// TIA Portal V19 export
DATA_BLOCK "JB"   // DB52
// stored: InstanceOfName JB_FB, InstanceOfType FB
"JB_FB"
   // VAR_INPUT
   //    AreaInterface : "AreaInterface";
   //    ZSI : "udt_ZoneSafetyInterface";
   //    DSI : Struct
   //       Torch : "udt_DeviceSafetyInterface";
   //       ClampEntry : "udt_DeviceSafetyInterface";
   //       ClampExit : "udt_DeviceSafetyInterface";
   //       CutHead : "udt_DeviceSafetyInterface";
   //       PinchRoll_Feed : "udt_DeviceSafetyInterface";
   //       PinchRoll_Lift : "udt_DeviceSafetyInterface";
   //    END_STRUCT;
   //    Drive : Struct
   //       Torch : "TAx_DriveInterface";
   //       Picnhroll_Feed : "TAx_DriveInterface";
   //    END_STRUCT;
   //    HWID : Struct
   //       Torch_TEL1 : HW_SUBMODULE;
   //       TorchEnc_IO : HW_SUBMODULE;
   //       Pinchroll_Feed_TEL1 : HW_SUBMODULE;
   //    END_STRUCT;
   //    DataIn : Struct
   //       WeldingCycle_AI_Potentiometer : Int;
   //       WeldingCycle_Pb_Stop : Bool;
   //       WeldingCycle_Pb_Start : Bool;
   //       WeldingCycle_Pb_StartStop : Bool;
   //       Welder_Pb_Man : Bool;
   //       CutHead_PbCycle : Bool;
   //       SAFETY_DeadMan_PB : Bool;
   //       Torch : "Positioning_DOL_Machine_DataIn";
   //       ClampEntry : "ValveMachine_DataIn";
   //       ClampExit : "ValveMachine_DataIn";
   //       CutHead : "ValveMachine_DataIn";
   //       PinchRoll_Feed : "SpeedMachine_DataIn";
   //       PinchRoll_Lift : "ValveMachine_DataIn";
   //    END_STRUCT;
   //    CIn : Struct
   //       Manager : "JB_Manager";
   //       PressureRunning : Bool;
   //    END_STRUCT;
   //    Config : Struct
   //       MeasurePasslineReference : Real;
   //       MaxMaterialWidth : Real;
   //       Torch : "Positioning_DOL_Machine_Config";
   //       ClampEntry : "ValveMachine_Config";
   //       ClampExit : "ValveMachine_Config";
   //       CutHead : "ValveMachine_Config";
   //       Pinchroll_Feed : "SpeedMachine_Config";
   //       Pinchroll_Lift : "ValveMachine_Config";
   //    END_STRUCT;
   // END_VAR
   // VAR_OUTPUT
   //    MachineInterface : "MachineInterface";
   //    DataOut : Struct
   //       LpWeldingCycle_1 : Bool;
   //       LpWeldingCycle_2 : Bool;
   //       WelderON : Bool;
   //       AspiratoreON : Bool;
   //       Torch : "Positioning_DOL_Machine_DataOut";
   //       ClampEntry : "ValveMachine_DataOut";
   //       ClampExit : "ValveMachine_DataOut";
   //       CutHead : "ValveMachine_DataOut";
   //       Pinchroll_Feed : "SpeedMachine_DataOut";
   //       Pinchroll_Lift : "ValveMachine_DataOut";
   //    END_STRUCT;
   //    COut : "JB_Status";
   // END_VAR
   // VAR_IN_OUT
   //    PersistentValues : Struct
   //       Data : Struct
   //          WeldingSetUp : "JB_WeldingSetUp";
   //          ClampEntryClosed : Bool;
   //          ClampExitClosed : Bool;
   //       END_STRUCT;
   //       Torch : Struct
   //          MeasureTorchHolder : LReal;
   //          InhibitWeld_Pos : LReal;
   //          InhibitWeld_Window : LReal;
   //          Parking_Pos : LReal;
   //          WeldingUseLocalData : Bool;
   //          Cycle_HighSpeed : LReal;
   //          Cycle_LowSpeed : LReal;
   //       END_STRUCT;
   //       TorchAx : "Positioning_DOL_Machine_Par";
   //       TorchAx_Pers : "Positioning_DOL_Machine_Pers_Data";
   //       TorchEnc : "PosFbk_RTN";
   //       PinchRoll_Feed : "SpeedMachine_Par";
   //       Aspiratore_TimeOff : Time;
   //    END_STRUCT;
   // END_VAR
   // VAR
   //    Alarm : Struct
   //       TorchAx : "Positioning_DOL_Machine_Alr";
   //       TorchEnc : "PosFbk_Encoder_Alr";
   //       ClampEntry : "ValveAlr";
   //       ClampExit : "ValveAlr";
   //       CutHead : "ValveAlr";
   //       Pinchroll_Feed : "SpeedMachine_Alr";
   //       Pinchroll_Lift : "ValveAlr";
   //    END_STRUCT;
   //    Warning : Struct
   //       TorchAx : "Positioning_DOL_Machine_Wng";
   //       ClampEntry : "ValveMachine_Wng";
   //       ClampExit : "ValveMachine_Wng";
   //       CutHead : "ValveMachine_Wng";
   //       Pinchroll_Feed : "SpeedMachine_Wng";
   //       Pinchroll_Lift : "ValveMachine_Wng";
   //    END_STRUCT;
   //    HMI : Struct
   //       Torch_B_Preset : Bool;
   //       Torch_PresetValue : LReal;
   //       Torch_FdbkPreset : LReal;
   //    END_STRUCT;
   //    Sts : Struct
   //       Torch : Struct
   //          InParkPosition : Bool;
   //          InOutEdgeOfWeldStart : Bool;
   //          InWeldStart : Bool;
   //          inWeldStop : Bool;
   //          InPotentimeterON : Bool;
   //          InWeldON : Bool;
   //          InWeldInhibit : Bool;
   //       END_STRUCT;
   //       WeldCycle : Struct
   //          Phase : Int;
   //          Cnd : Bool;
   //          ON1 : Bool;
   //          ON2 : Bool;
   //          PercentagePotentiometer : Real;
   //          PosOutStripEdgeSideWeldStart : LReal;
   //          PosOutStripEdgeSideWeldStop : LReal;
   //          PosStripEdgeSideWeldStart : LReal;
   //          PosStripEdgeSideWeldStop : LReal;
   //          PosWeldStart : LReal;
   //          PosWeldStop : LReal;
   //          PosMinusInhibit : LReal;
   //          PosPlusInhibit : LReal;
   //          TON_Pause { S7_SetPoint := 'True'} : TON_TIME;
   //       END_STRUCT;
   //       CutCycle : Struct
   //          ON : Bool;
   //          OK_Rest : Bool;
   //          OK_Work : Bool;
   //       END_STRUCT;
   //    END_STRUCT;
   //    Ctrl : Struct
   //       WeldCycle : Struct
   //          Clamps_Close : Bool;
   //          Clamps_Open : Bool;
   //          Welder_ON : Bool;
   //          Torch_MoveToPos_Park : Bool;
   //          Torch_MoveToPos_Start : Bool;
   //          Torch_MoveToPos_StartBack : Bool;
   //          Torch_VelBwd_WeldON : Bool;
   //          Torch_VelFwd_WeldON : Bool;
   //       END_STRUCT;
   //       Welder : Struct
   //          Man_ON : Bool;
   //       END_STRUCT;
   //    END_STRUCT;
   //    Torch : "Positioning_DOL_Machine_FB";
   //    TorchEnc : "PosFbk_SickANM58";
   //    TorchEncITF : "PosFbk_ITF";
   //    ClampEntry : "ValveMachine_FB";
   //    ClampExit : "ValveMachine_FB";
   //    CutHead : "ValveMachine_FB";
   //    PinchRoll_Feed : "SpeedMachine_FB";
   //    PinchRoll_Lift : "ValveMachine_FB";
   //    TON_LiftPbUp : TON_TIME;
   //    TOF_Aspiratore { S7_SetPoint := 'True'} : TOF_TIME;
   //    AUX : Struct
   //       PbStartStop { ExternalAccessible := 'False'; ExternalVisible := 'False'; ExternalWritable := 'False'} : Bool;
   //       PbStart2 : Bool;
   //       Welder_Pb_Man : Bool;
   //       UseDataPPrf : Bool;
   //       Weld_PbCycle : Bool;
   //       Cut_PbCycle : Bool;
   //    END_STRUCT;
   // END_VAR
BEGIN
END_DATA_BLOCK
